FUNCTION_BLOCK bfb_ess_battery
  (* Standard: 61499-2 *)
  (* Version 0.1, 2018-00-07, hpea485, UOA *)
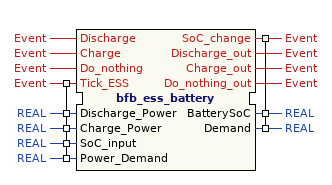
  EVENT_INPUT
    Discharge;
    Charge;
    Do_nothing;
    Tick_ESS WITH Discharge_Power, Charge_Power, SoC_input, Power_Demand;
  END_EVENT
  EVENT_OUTPUT
    SoC_change WITH BatterySoC, Demand;
    Discharge_out;
    Charge_out;
    Do_nothing_out;
  END_EVENT
  VAR_INPUT
    Discharge_Power : REAL;
    Charge_Power : REAL := 1;
    SoC_input : REAL;
    Power_Demand : REAL;
  END_VAR
  VAR_OUTPUT
    BatterySoC : REAL;
    Demand : REAL;
  END_VAR
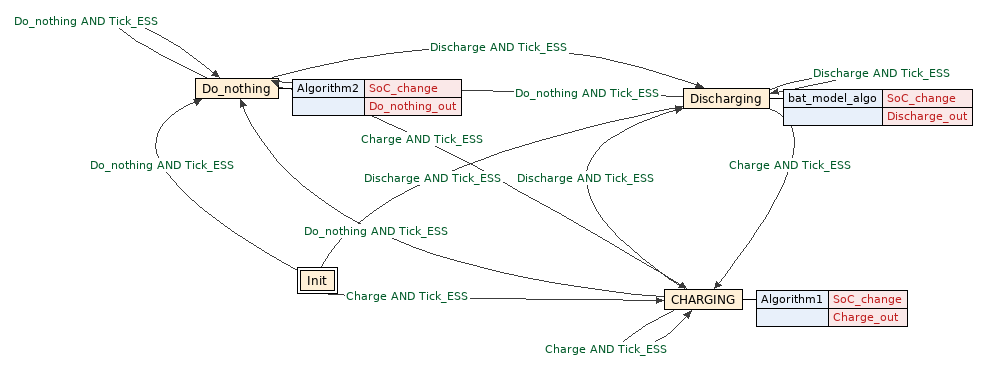
  EC_STATES
    Init;
    Do_nothing : Algorithm2 -> SoC_change, -> Do_nothing_out;
    Discharging : bat_model_algo -> SoC_change, -> Discharge_out;
    CHARGING : Algorithm1 -> SoC_change, -> Charge_out;
  END_STATES
  EC_TRANSITIONS
    Do_nothing TO Discharging := Discharge AND Tick_ESS;
    Do_nothing TO CHARGING := Charge AND Tick_ESS;
    Do_nothing TO Do_nothing := Do_nothing AND Tick_ESS;
    Discharging TO CHARGING := Charge AND Tick_ESS;
    Discharging TO Do_nothing := Do_nothing AND Tick_ESS;
    Discharging TO Discharging := Discharge AND Tick_ESS;
    CHARGING TO Discharging := Discharge AND Tick_ESS;
    CHARGING TO Do_nothing := Do_nothing AND Tick_ESS;
    CHARGING TO CHARGING := Charge AND Tick_ESS;
    Init TO Do_nothing := Do_nothing AND Tick_ESS;
    Init TO CHARGING := Charge AND Tick_ESS;
    Init TO Discharging := Discharge AND Tick_ESS;
  END_TRANSITIONS
  ALGORITHM bat_model_algo IN C:
REAL SoC = me->SoC_input;
REAL discharge = me->Discharge_Power;
REAL cb = 620;// kwh from Kalpesh code, power required by ESS to charge 100% in 1 hour i.e 1C rate
REAL Demand = me->Power_Demand;
me->Demand = Demand;

me->BatterySoC = SoC - (discharge*100/(cb*60));
SoC = SoC - (discharge*100/(cb*60));
printf("SoC_discharge : %f  \r\n",me->BatterySoC);

//Have better modelling
//current_SoC += me->Minutes_per_tick * me->Current_A; //WRONG: Fix

//#define MAX_SOC 100
//#define MIN_SOC 0

//if(current_SoC > MAX_SOC) {
	//current_SoC = MAX_SOC;
//} else if (current_SoC < MIN_SOC) {
	//current_SoC = MIN_SOC;
//}

//me->Current_SoC = current_SoC;
  END_ALGORITHM
  ALGORITHM Algorithm1 IN C:
REAL SoC = me->SoC_input;
REAL charge = me->Charge_Power;
REAL Demand = me->Power_Demand;
me->Demand = Demand;

REAL cb = 620;// kwh from Kalpesh code, power required by ESS to charge 100% in 1 hour i.e 1C rate
me->BatterySoC = SoC + charge*100/(cb*60);
SoC = SoC + charge*100/(cb*60);
printf("SoC_charge : %f  \r\n",me->BatterySoC);
  END_ALGORITHM
  ALGORITHM Algorithm2 IN C:
//static REAL SoC = 0;
printf("welcome to soc initial \r\n");
me->BatterySoC = me->SoC_input;

REAL Demand = me->Power_Demand;
me->Demand = Demand;
printf("power : %f, %f \r\n", Demand, me->Power_Demand);
  END_ALGORITHM
END_FUNCTION_BLOCK
